{attribute 'GeneratedUsingTerminal: EL6090-0000-0016'}
{attribute addProperty BoxType "EL6090-0000-0016"}
{attribute addProperty Id "Value_rowAT %Q*ARRAY[0..1] OF INT4"}
{attribute addProperty CRC "4003442326"}
{attribute addProperty Size "4"}
TYPE DIS_Outputs_6C9BFFEE :
STRUCT
	{attribute addProperty Name "Value_row"}
	Value_row AT %Q* : ARRAY[0..1] OF INT;
END_STRUCT
END_TYPE

(* stored: Version 1.2.0.0, ProductVersion 3.1.4024.9
   DUT DIS_Outputs_6C9BFFEE: Id {6832fea1-b807-4e98-ad21-fb71606fbca8} *)
